(* PLC project Trafic_Light, Unknown Unnamed 1 *)
(* stored: creationDateTime 2020-10-12T21:33:17, modificationDateTime 2022-08-17T11:38:55 *)

PROGRAM Trafic_light
  VAR
    TOF0 : TOF;
    TOF1 : TOF;
    TOF2 : TOF;
  END_VAR
  VAR
    O_LEDRed AT %QX0.0 : BOOL;  (* This can be a red LED on pin 7 *)
    O_LEDOrange AT %QX0.1 : BOOL;  (* This can be a orange LED on pin 8 *)
    O_LEDGreen AT %QX0.2 : BOOL;  (* This can be a Green LED on pin 12 *)
    First_cycle AT %QX0.3 : BOOL := TRUE;  (* Is true only during the first scan cycle *)
  END_VAR
  VAR
    F_TRIG0 : F_TRIG;
    F_TRIG1 : F_TRIG;
    F_TRIG2 : F_TRIG;
  END_VAR

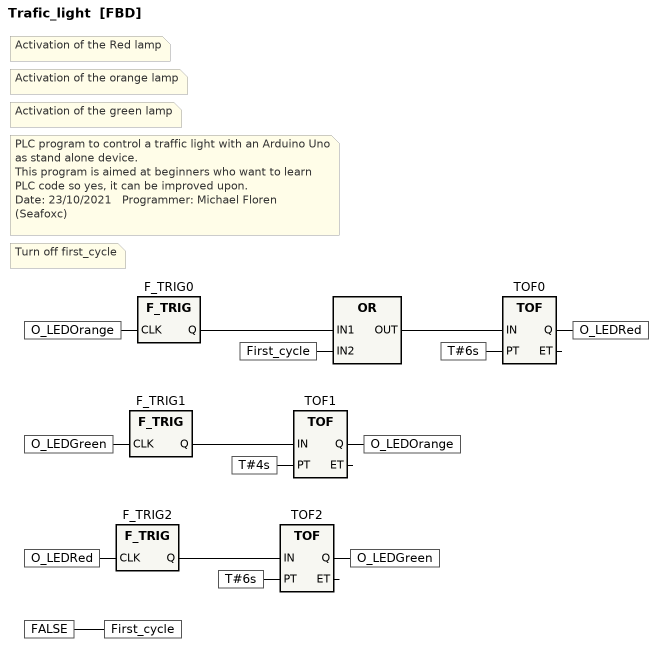
(* FBD diagram, written out as Structured Text *)
(* PLC program to control a traffic light with an Arduino Uno as stand alone device.
This program is aimed at beginners who want to learn PLC code so yes, it can be improved upon. 

Date: 23/10/2021   Programmer: Michael Floren  (Seafoxc) *)
(* Activation of the Red lamp *)
F_TRIG0(CLK := O_LEDOrange);
TOF0(IN := F_TRIG0.Q OR First_cycle, PT := T#6s);
O_LEDRed := TOF0.Q;
(* Activation of the orange lamp *)
F_TRIG1(CLK := O_LEDGreen);
TOF1(IN := F_TRIG1.Q, PT := T#4s);
O_LEDOrange := TOF1.Q;
(* Activation of the green lamp *)
F_TRIG2(CLK := O_LEDRed);
TOF2(IN := F_TRIG2.Q, PT := T#6s);
O_LEDGreen := TOF2.Q;
(* Turn off first_cycle *)
First_cycle := FALSE;
END_PROGRAM

CONFIGURATION Config0
  RESOURCE Res0 ON PLC
    TASK task0(INTERVAL := T#20ms, PRIORITY := 0);
    PROGRAM instance0 WITH task0 : Trafic_light;
  END_RESOURCE
END_CONFIGURATION
